FUNCTION_BLOCK FB_CsvPersistentEventStorage IMPLEMENTS I_PersistentEventStorage
VAR
	fbFileOpen : FB_FileOpen := (sPathName := 'C:\Events.log', nMode := FOPEN_MODEAPPEND OR FOPEN_MODETEXT);
	fbFilePuts : FB_FilePuts;
    fbFileClose : FB_FileClose;
   	eWriteState : (WAIT_FOR_EVENT,FILE_OPEN_TRIGGER, FILE_OPEN,   WRITE_EVENT_TRIGGER, WRITE_EVENT, FILE_CLOSE_TRIGGER ,FILE_CLOSE, ERROR);
	stEventWrittenToFile : ST_Event;
	
	CsvString : T_MaxString;
END_VAR

CASE eWriteState OF
	FILE_OPEN_TRIGGER :
		fbFileOpen(bExecute := TRUE);
		eWriteState := FILE_OPEN;
		
	FILE_OPEN :
	    fbFileOpen(bExecute := FALSE);
		IF fbFileOpen.bError THEN
			eWriteState := ERROR;
		ELSIF NOT fbFileOpen.bBusy AND fbFileOpen.hFile <> 0 THEN
			eWriteState := WAIT_FOR_EVENT;
		END_IF
		
    WAIT_FOR_EVENT :
      //DO Nothing
	  
	WRITE_EVENT_TRIGGER:
	  CsvString := CreateCsvString(stEvent := stEventWrittenToFile);
	fbFilePuts(bExecute := TRUE, sLine := CsvString, hFile :=fbFileOpen.hFile);
	eWriteState := WRITE_EVENT;  
	
    WRITE_EVENT: 
	 fbFilePuts(bExecute := FALSE);
	   
	IF fbFilePuts.bError THEN 
		eWriteState:= ERROR;
	ELSIF NOT fbFilePuts.bBusy THEN 
		eWriteState := FILE_CLOSE_TRIGGER;
	END_IF
	
	FILE_CLOSE_TRIGGER:
	fbFileClose(bExecute := TRUE, hFile :=fbFileOpen.hFile);
    eWriteState := FILE_CLOSE;
	
    FILE_CLOSE:
	//CLOSE THE FILE
	fbFileClose(bExecute := FALSE);
	IF fbFileClose.bError THEN
		eWriteState := ERROR;
	ELSIF NOT fbFileClose.bBusy THEN
		eWriteState := FILE_OPEN_TRIGGER;
	END_IF
	
	ERROR : 
	//Do Nothing
	
END_CASE

METHOD PRIVATE CreateCsvString :T_MaxString
VAR_INPUT
	stEvent : REFERENCE TO ST_Event;
END_VAR
VAR
	TempString : T_MaxString;
END_VAR
TempString := TO_STRING(stEvent.eEventType);
TempString := CONCAT(STR1 :=TempString , STR2 :=', ');
TempString := CONCAT(STR1 :=TempString , STR2 := TO_STRING(stEvent.eEventSeverity));
TempString := CONCAT(STR1 :=TempString , STR2 :=', ');
TempString := CONCAT(STR1 :=TempString , STR2 := TO_STRING(stEvent.nEventIdentity));
TempString := CONCAT(STR1 :=TempString , STR2 :=', ');
TempString := CONCAT(STR1 :=TempString , STR2 :=TO_STRING(stEvent.sEventText));
TempString := CONCAT(STR1 :=TempString , STR2 :=', ');
TempString := CONCAT(STR1 :=TempString , STR2 :=TO_STRING(stEvent.dtTimeStamp));
TempString := CONCAT(STR1 :=TempString , STR2 :='$n');

CreateCsvString := TempString;
END_METHOD


METHOD StoreEvent
VAR_INPUT
	stEvent	: ST_Event;
END_VAR
IF eWriteState = WAIT_FOR_EVENT THEN
	eWriteState := WRITE_EVENT_TRIGGER;
	stEventWrittenToFile := stEvent;
END_IF
END_METHOD

END_FUNCTION_BLOCK

(* stored: Version 1.1.0.1, ProductVersion 3.1.4024.16
   POU FB_CsvPersistentEventStorage: Id {4f3b813b-ede0-49ce-baca-e9a65872a1a9}, SpecialFunc None
   Method CreateCsvString: Id {04e8714c-9653-4763-83fd-5baee407507e}
   Method StoreEvent: Id {a8f04c63-2584-4039-99ec-4b58ccc301a1} *)
